(* PLC project test3 HCFA_Q1 optional.project, CODESYS CODESYS V3.5 SP14 Patch 1 *)
(* stored: creationDateTime 2026-10-07T21:32:52.8166491, modificationDateTime 2026-10-07T21:17:46.3844832 *)

TYPE ST_A6Control : STRUCT
  Control_word : U_A6ControlWord;  (* 6040h - Управляющее слово *)
  Target_position : DINT;  (* 607Ah - Целевая позиция *)
  Target_velocity : DINT;  (* 60FFh - Целевая скорость *)
  Target_torque : INT;  (* 6071h - Целевой момент *)
  Modes_of_operation : E_ModesOfOperation;  (* 6060h - Режим работы (SINT!) *)
  Touch_probe_function : U_A6TouchProbeFunction;  (* 60B8h - Функция Touch Probe *)
  Max_profile_velocity : UDINT;  (* 607Fh - Макс. скорость профиля *)
  Positive_torque_limit : UINT;  (* 60E0h - Положительный лимит момента *)
  Negative_torque_limit : UINT;  (* 60E1h - Отрицательный лимит момента *)
END_STRUCT;
END_TYPE

TYPE ST_A6Status : STRUCT
  Error_code : E_ErrorCode;  (* 603Fh - Код ошибки *)
  Statusword : U_A6StatusWord;  (* 6041h - Статусное слово *)
  Position_actual_value : DINT;  (* 6064h - Фактическая позиция *)
  Torque_actual_value : INT;  (* 6077h - Фактический момент *)
  Modes_of_operation_disp : E_ModesOfOperation;  (* 6061h - Отображение режима работы *)
  Following_error_actual : DINT;  (* 60F4h - Фактическое рассогласование *)
  Touch_probe_status : U_A6TouchProbeStatus;  (* 60B9h - Статус Touch Probe *)
  Touch_probe_pos1_value : DINT;  (* 60BAh - Значение Touch Probe 1 *)
  Touch_probe_pos2_value : DINT;  (* 60BCh - Значение Touch Probe 2 *)
  Velocity_actual_value : DINT;  (* 606Ch - Фактическая скорость *)
END_STRUCT;
END_TYPE

TYPE ST_A6 : STRUCT
  In : ST_A6Status;
  Out : ST_A6Control;
END_STRUCT;
END_TYPE

TYPE HW_ALL : STRUCT
  DI : DI;
  Dout : Dout;
  AI : AI;
  Servo : Servo;
END_STRUCT;
END_TYPE

TYPE DI : STRUCT

END_STRUCT;
END_TYPE

TYPE Dout : STRUCT

END_STRUCT;
END_TYPE

TYPE AI : STRUCT

END_STRUCT;
END_TYPE

TYPE AO : STRUCT

END_STRUCT;
END_TYPE

TYPE Servo : STRUCT
  Axis_Move : ST_A6;
  Axis_UP_Left : ST_A6;
  Axis_UP_Right : ST_A6;
END_STRUCT;
END_TYPE

(* values of E_ModesOfOperation: No_Mode: Режим не задан; PP: Profile Position; PV: Profile Velocity; PT: Profile Torque; HM: Homing Mode; CSP: Cyclic Synchronous Position; CSV: Cyclic Synchronous Velocity; CST: Cyclic Synchronous Torque *)

{attribute 'qualified_only'}
{attribute 'strict'}
TYPE E_ModesOfOperation : (No_Mode := 0, PP := 1, PV := 3, PT := 4, HM := 6, CSP := 8, CSV := 9, CST := 10);
END_TYPE

TYPE ST_ControlWord_Bits : STRUCT
  Switch_on : BIT;  (* Бит 0 *)
  Enable_voltage : BIT;  (* Бит 1 *)
  Quick_stop : BIT;  (* Бит 2 (0 = Quick stop active) *)
  Enable_operation : BIT;  (* Бит 3 *)
  Op_mode_specific_1 : BIT;  (* Бит 4 (New set-point / Enable ramp) *)
  Op_mode_specific_2 : BIT;  (* Бит 5 (Change set immediately / Unlock ramp) *)
  Op_mode_specific_3 : BIT;  (* Бит 6 (Absolute / Relative) *)
  Fault_reset : BIT;  (* Бит 7 (0->1 = Reset fault) *)
  Halt : BIT;  (* Бит 8 *)
  Op_mode_specific_4 : BIT;  (* Бит 9 *)
  Reserved_10 : BIT;  (* Бит 10 *)
  Manufacturer_1 : BIT;  (* Бит 11 *)
  Manufacturer_2 : BIT;  (* Бит 12 *)
  Manufacturer_3 : BIT;  (* Бит 13 *)
  Manufacturer_4 : BIT;  (* Бит 14 *)
  Manufacturer_5 : BIT;  (* Бит 15 *)
END_STRUCT;
END_TYPE

TYPE ST_StatusWord_Bits : STRUCT
  Ready_to_switch_on : BIT;  (* Бит 0 *)
  Switched_on : BIT;  (* Бит 1 *)
  Operation_enabled : BIT;  (* Бит 2 *)
  Fault : BIT;  (* Бит 3 *)
  Voltage_enabled : BIT;  (* Бит 4 *)
  Quick_stop : BIT;  (* Бит 5 (0 = Quick stop active) *)
  Switch_on_disabled : BIT;  (* Бит 6 *)
  Warning : BIT;  (* Бит 7 *)
  Manufacturer_1 : BIT;  (* Бит 8 *)
  Remote : BIT;  (* Бит 9 *)
  Target_reached : BIT;  (* Бит 10 (Position/Speed/Torque reached) *)
  Internal_limit_active : BIT;  (* Бит 11 *)
  Op_mode_specific_1 : BIT;  (* Бит 12 (Set-point acknowledge / Speed) *)
  Op_mode_specific_2 : BIT;  (* Бит 13 (Following error) *)
  Manufacturer_2 : BIT;  (* Бит 14 *)
  Manufacturer_3 : BIT;  (* Бит 15 *)
END_STRUCT;
END_TYPE

(* values of E_ErrorCode: No_Error: ================= Нет ошибки =================; Er01_0_SW_Version_Mismatch: ================= Class 1: Non-resettable ================= --- Ошибки версий и параметров ---; Er05_0_Current_Loop_Timeout: --- Ошибки таймаутов циклов ---; Er06_0_Runaway_Protection: --- Защита от разгона ---; Er10_0_P_HW_Overcurrent: --- Токовые ошибки ---; Er11_0_Excessive_Motor_Speed_PowerOn: --- Ошибки мотора ---; Er20_1_Encoder_Internal_Fault: --- Ошибки энкодера ---; Er31_0_More_Than_10_PDO_Objects: --- Ошибки EtherCAT ---; Er40_0_Drive_Overload: ================= Class 1: Resettable =================; Er80_0_Control_Power_Undervoltage: ================= Class 2 (Предупреждения) =================; ALF0_0_Emergency_Stop_Alarm: ================= Class 3: Alarms (Алармы) ================= *)

{attribute 'qualified_only'}
{attribute 'strict'}
TYPE E_ErrorCode : (No_Error := 16#0, Er01_0_SW_Version_Mismatch := 16#100, Er01_1_Motor_Param_Mismatch := 16#110, Er02_0_No_Drive_Match := 16#200, Er02_1_No_Motor_Match := 16#210, Er02_2_No_Encoder_Match := 16#220, Er03_0_System_Param_Error := 16#300, Er03_1_Param_Out_of_Range := 16#310, Er03_2_Param_Write_Error := 16#320, Er03_3_Param_Read_Error := 16#330, Er05_0_Current_Loop_Timeout := 16#500, Er05_1_Speed_Loop_Timeout := 16#510, Er05_2_Position_Loop_Timeout := 16#520, Er05_3_Serial_Data_Check_Fail := 16#530, Er06_0_Runaway_Protection := 16#600, Er10_0_P_HW_Overcurrent := 16#1000, Er10_1_N_HW_Overcurrent := 16#1010, Er10_2_U_SW_Overcurrent := 16#1020, Er10_3_V_SW_Overcurrent := 16#1030, Er10_4_Output_Short_to_Ground := 16#1040, Er10_5_Current_Sampling_Fail := 16#1050, Er10_6_Incorrect_Current_Param := 16#1060, Er10_7_UV_Current_Correction_Fail := 16#1070, Er10_8_Excessive_Current_Zero_Drift := 16#1080, Er10_9_Current_Exception_Enabling := 16#1090, Er11_0_Excessive_Motor_Speed_PowerOn := 16#1100, Er11_1_Drive_Over_Temperature := 16#1110, Er20_1_Encoder_Internal_Fault := 16#2010, Er20_2_Encoder_Read_Write_Error := 16#2020, Er20_3_Encoder_Data_Frame_Loss := 16#2030, Er20_4_Encoder_Incremental_Overflow := 16#2040, Er20_5_Abnormal_Encoder_Data := 16#2050, Er20_6_Encoder_Type_Mismatch := 16#2060, Er20_7_Encoder_Model_Unsupported := 16#2070, Er20_8_Encoder_Battery_Failure := 16#2080, Er20_9_Encoder_MultiTurn_Error := 16#2090, Er21_0_Encoder_Pulse_Mismatch := 16#2100, Er31_0_More_Than_10_PDO_Objects := 16#3100, Er32_0_EtherCAT_Peripheral_Error := 16#3200, Er32_1_ESI_Check_Error := 16#3210, Er32_2_EEPROM_Read_Fail := 16#3220, Er32_3_EEPROM_Update_Fail := 16#3230, Er32_4_ESC_Checksum_Error := 16#3240, Er32_5_XML_Info_Fail := 16#3250, Er40_0_Drive_Overload := 16#4000, Er41_0_Motor_Overload := 16#4100, Er41_1_Motor_Locked_Rotor := 16#4110, Er41_2_Motor_Over_Temperature := 16#4120, Er42_1_Discharge_Tube_Temp_High := 16#4210, Er42_2_Heatsink_Temp_High := 16#4220, Er43_0_Overvoltage := 16#4300, Er43_1_Undervoltage := 16#4310, Er45_0_S_ON_Enabling_Failure := 16#4500, Er46_0_Motor_Overspeed := 16#4600, Er47_0_Excessive_Position_Deviation := 16#4700, Er47_1_Position_Deviation_Overflow := 16#4710, Er50_1_DQ_Current_Overflow := 16#5010, Er51_0_Offline_Inertia_AutoTune_Fail := 16#5100, Er51_1_Offline_Inertia_Param_Error := 16#5110, Er52_0_Angle_AutoTuning_Failure := 16#5200, Er53_0_Motor_Param_AutoTune_Timeout := 16#5300, Er53_1_Resistance_AutoTune_Fail := 16#5310, Er53_2_Inductance_AutoTune_Fail := 16#5320, Er53_3_BackEMF_AutoTune_Fail := 16#5330, Er54_0_Current_Loop_AutoTune_Fail := 16#5400, Er55_0_Excessive_Vibration := 16#5500, Er74_0_EtherCAT_Sync_Cycle_Error := 16#7400, Er74_1_No_Sync_Signal := 16#7410, Er74_2_Chip_Sync_Incomplete_OP := 16#7420, Er80_0_Control_Power_Undervoltage := 16#8000, Er81_0_Input_Phase_Loss_1 := 16#8100, Er81_1_Input_Phase_Loss_2 := 16#8110, Er81_2_Output_Phase_Loss := 16#8120, Er82_0_DI_Function_Allocation_Fault := 16#8200, Er82_1_DO_Function_Allocation_Fault := 16#8210, Er84_0_Electronic_Gear_Ratio_Error := 16#8400, Er84_1_Software_Limit_Setting_Error := 16#8410, Er84_2_Encoder_Resolution_Error := 16#8420, Er84_3_Home_Position_Setting_Error := 16#8430, Er87_1_OneTime_Pos_Ref_Increment := 16#8710, Er87_2_Continuous_Pos_Ref_Increment := 16#8720, Er87_3_Target_Pos_32bit_Overflow := 16#8730, Er87_4_Target_Pos_Exceeds_SingleTurn := 16#8740, ErA0_1_MultiTurn_Overflow_Fault := 16#A010, ErC1_0_EtherCAT_Sync_Period_Error := 16#C100, ErC1_1_Synchronization_Loss := 16#C110, ErC1_2_Network_Status_Switch_Error := 16#C120, ErC1_4_Network_Cable_Unreliable := 16#C140, ErC1_5_Data_Frame_Loss_Protection := 16#C150, ErC1_6_Data_Frame_Forwarding_Error := 16#C160, ErC1_7_Data_Update_Timeout := 16#C170, ErC1_8_Watchdog_Expired := 16#C180, ErC2_0_SYNC_Signal_Loss := 16#C200, ALF0_0_Emergency_Stop_Alarm := 16#F000, ALF1_0_RePowerOn_Required := 16#F100, ALF1_1_Frequent_Param_Storage_Alarm := 16#F110, ALF1_2_Torque_Reached_Param_Error := 16#F120, ALF1_3_Too_Frequent_EEPROM_Writing := 16#F130, ALF2_0_Forward_Overtravel_Alarm := 16#F200, ALF2_1_Reverse_Overtravel_Alarm := 16#F210, ALF4_0_Homing_Timeout := 16#F400, ALF4_1_Homing_DI_Conflict := 16#F410, ALF4_2_Homing_Mode_Conflict := 16#F420, ALF5_0_Braking_Resistor_Overload := 16#F500, ALF5_1_External_Brake_Resistance_Low := 16#F510, ALF6_1_Output_Phase_Loss := 16#F610, ALF8_0_Vibration_During_AutoTuning := 16#F800, ALF9_0_Encoder_Battery_Voltage_Low := 16#F900, ALFA_0_Drive_High_Temp_Warning := 16#FAA0, xxnr_Servo_Not_Ready := 16#FFFF) UINT;
END_TYPE

TYPE ST_TouchProbeStatus_Bits : STRUCT

END_STRUCT;
END_TYPE

TYPE ST_TouchProbeFunction_Bits : STRUCT
  TP1_Enable : BIT;  (* Бит 0: 0=Disabled, 1=Enabled *)
  TP1_TriggerMode : BIT;  (* Бит 1: 0=Single, 1=Continuous *)
  TP1_SignalSource : BIT;  (* Бит 2: 0=DI signal, 1=Z signal *)
  Reserved_3 : BIT;  (* Бит 3 *)
  TP1_PosEdge_Enable : BIT;  (* Бит 4: Разрешить захват по положительному фронту *)
  TP1_NegEdge_Enable : BIT;  (* Бит 5: Разрешить захват по отрицательному фронту *)
  Reserved_6 : BIT;  (* Бит 6 *)
  Reserved_7 : BIT;  (* Бит 7 *)
  TP2_Enable : BIT;  (* Бит 8 *)
  TP2_TriggerMode : BIT;  (* Бит 9 *)
  TP2_SignalSource : BIT;  (* Бит 10 *)
  Reserved_11 : BIT;  (* Бит 11 *)
  TP2_PosEdge_Enable : BIT;  (* Бит 12 *)
  TP2_NegEdge_Enable : BIT;  (* Бит 13 *)
  Reserved_14 : BIT;  (* Бит 14 *)
  Reserved_15 : BIT;  (* Бит 15 *)
END_STRUCT;
END_TYPE

PROGRAM PLC_PRG

END_PROGRAM

PROGRAM PLC_PRG

          //Qumark:=GVL.Qumark;
    
        
END_PROGRAM

CONFIGURATION Device
  RESOURCE Application ON PLC
    {attribute 'qualified_only'}
    VAR_GLOBAL  (* HW *)
      IO : HW_ALL;
    END_VAR
    TASK MainTask(INTERVAL := T#4ms, PRIORITY := 1);
    TASK EtherCAT_Task(INTERVAL := T#4ms, PRIORITY := 1);
    TASK VISU_TASK(INTERVAL := T#100ms, PRIORITY := 31);
    PROGRAM PLC_PRG WITH MainTask : PLC_PRG;
    PROGRAM VisuElems.Visu_Prg WITH VISU_TASK : VisuElems.Visu_Prg;
  END_RESOURCE
END_CONFIGURATION

CONFIGURATION LocalDevice
END_CONFIGURATION

CONFIGURATION GeneralIO
END_CONFIGURATION

CONFIGURATION SoftMotion General Axis Pool
END_CONFIGURATION

CONFIGURATION Ethernet
END_CONFIGURATION

CONFIGURATION EtherCAT_Master_SoftMotion
END_CONFIGURATION

CONFIGURATION LocalEtherCATDevice
END_CONFIGURATION

CONFIGURATION A6N_Servo_Driver
END_CONFIGURATION
